INTERFACE I_HostStructureMembers EXTENDS __SYSTEM.IQueryInterface

PROPERTY PUBLIC Members : I_StructureMembers
GET
END_GET
END_PROPERTY

END_INTERFACE

(* stored: Version 1.1.0.1, ProductVersion 3.1.4024.12
   Itf I_HostStructureMembers: Id {b619b8ab-031f-0bf8-1d3e-d3d064db4508}
   Property Members: Id {c5e81104-ef06-454c-80cf-dc98734595cd}
   Get Get: Id {f4b25703-1c06-4277-9e64-a25639db9fbf} *)
